FUNCTION F_TargetReachedOrLower : BOOL
VAR_INPUT
	fCurrentPos: LREAL;
	fTargetPos: LREAL;
END_VAR


F_TargetReachedOrLower := fCurrentPos <= (fTargetPos + fEpsilon);

END_FUNCTION

(* stored: Version 1.1.0.1, ProductVersion 3.1.4022.9
   POU F_TargetReachedOrLower: Id {2b97017a-3965-41d7-b115-f4a1b992fc4e}, SpecialFunc None *)
